TYPE ST_CHM_GenericHierarchy :
STRUCT
	HierarchyType		:	STRING(5);
	PerformedAction	:	STRING(10);
	TrackingLevels		:	STRING(10);
	TrackingIndicator	:	STRING(3);
	CaseItem			:	ST_CaseItem;

END_STRUCT
END_TYPE

(* stored: Version 1.1.0.1
   DUT ST_CHM_GenericHierarchy: Id {16378c5c-a042-4952-ae53-d580288ec9d2} *)
